Fanuc KAREL source: kt00799.KL

PROGRAM KT00799
%NOLOCKGROUP
VAR
R1:REAL;R2:REAL;OUT:REAL
BEGIN
--
--
R1=2.0
R2=3.0
R1=2.0
R2=3.0
OUT=EXP(R1)
END KT00799
